FUNCTION_BLOCK Light IMPLEMENTS I_LIGHT

VAR
	Output AT %Q* : BOOL;
END_VAR

METHOD Off
Output := FALSE;
END_METHOD

METHOD On
Output := TRUE;
END_METHOD

END_FUNCTION_BLOCK

(* stored: Version 1.1.0.1, ProductVersion 3.1.4024.12
   POU Light: Id {b25df339-94d3-426f-8e7f-5b55729b3085}, SpecialFunc None
   Method Off: Id {aeeae483-b9c9-44b1-90c3-e0e30d82e26e}
   Method On: Id {ca8880a9-66d8-4f04-930a-a751876446b3} *)
